FUNCTION TryConvert_TIME_TO_STRING : BOOL
VAR_INPUT
	in : TIME;
	out : REFERENCE TO STRING;
END_VAR

out := TIME_TO_STRING(in);
TryConvert_TIME_TO_STRING := TRUE;

END_FUNCTION

(* stored: Version 1.1.0.1, ProductVersion 3.1.4024.12
   POU TryConvert_TIME_TO_STRING: Id {d4a5aab7-60c0-4d70-bafd-f7a8f958ecce}, SpecialFunc None *)
